FUNCTION TFClearWorkAreaBCRead : BOOL
VAR_INPUT
	WorkAreaState : POINTER TO TFMachinePalletizer_WorkAreaState;
END_VAR
VAR
	i : INT;
END_VAR

FOR i:=1 TO MAXNUMBARCODE DO
	WorkAreaState^.BCRead[i].State := LETTURA_ESEGUITA;
	WorkAreaState^.BCRead[i].Value := ''; 
	WorkAreaState^.BCRead[i].ErrorCode := 0;
END_FOR
TFClearWorkAreaBCRead := TRUE;

END_FUNCTION

(* stored: Version 1.1.0.1, ProductVersion 3.1.4024.11
   POU TFClearWorkAreaBCRead: Id {18677100-7f80-4335-9682-3d0a85ada434}, SpecialFunc None *)
